(* PLC project  *)

CONFIGURATION Empty_Module_1
END_CONFIGURATION
